{attribute addProperty BoxType "EP9576-1032-0016"}
{attribute addProperty Id "BCT_InputsAT %I*BCT_Inputs_4FFA390D136170WcStateAT %I*WcState_F855686C1620InfoDataAT %I*InfoData_BC63D37F80100"}
{attribute addProperty CRC "2937750143"}
{attribute addProperty SizeInBites "232"}
{attribute addProperty SizeInBytes "29"}
TYPE EP9576_B5DF83EF :
STRUCT
	{attribute addProperty Name "BCT_Inputs"}
	BCT_Inputs : BCT_Inputs_4FFA390D;
	{attribute addProperty Name "WcState"}
	WcState : WcState_F855686C;
	{attribute addProperty Name "InfoData"}
	InfoData : InfoData_BC63D37F;
END_STRUCT
END_TYPE

(* stored: Version 1.2.0.0, ProductVersion 3.1.4024.9
   DUT EP9576_B5DF83EF: Id {df3f6a06-430a-4392-a5f6-2fe86326dcc6} *)
